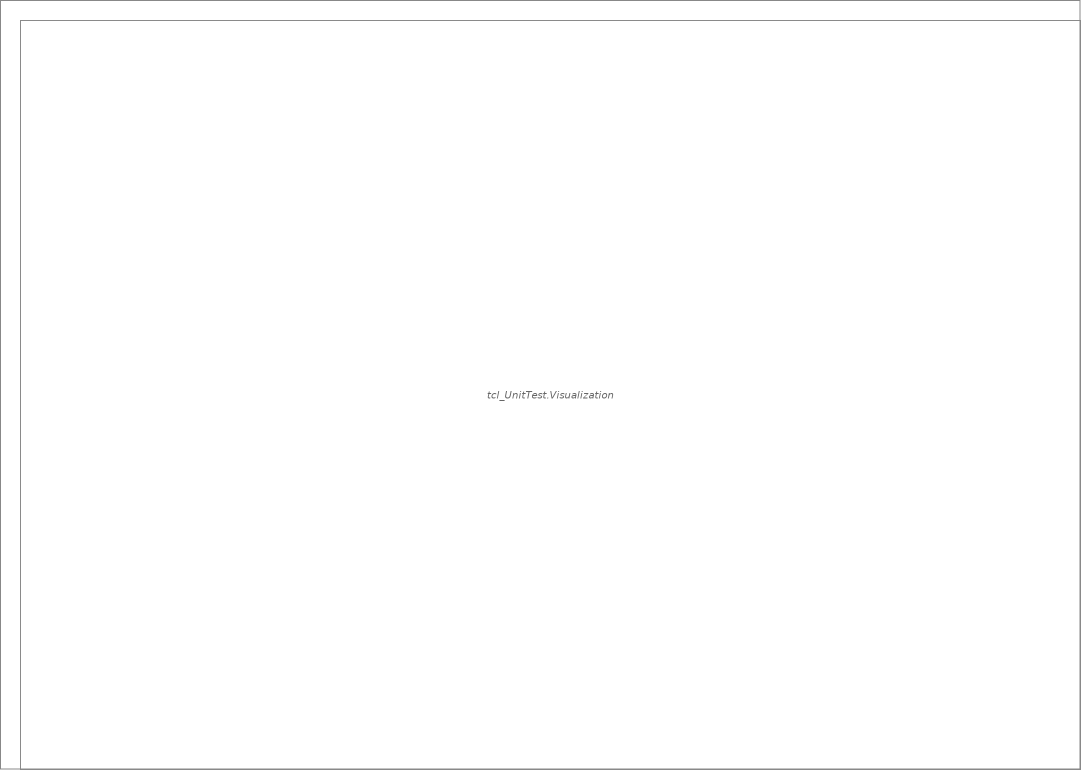
VISUALIZATION Visualization  // 1081x770
    Frame (20,20 1061x750)
        shows tcl_UnitTest.Visualization()
END_VISUALIZATION

(* stored: Version 1.1.0.1, ProductVersion 3.1.4024.3
   Visu Visualization: Id {2e451101-17d5-07f2-2e59-0982195421c1} *)
